FUNCTION IsValidExtension : BOOL
VAR_INPUT
	Extension : I_Extension;
END_VAR

IsValidExtension := Extension <> 0;

END_FUNCTION

(* stored: Version 1.1.0.1, ProductVersion 3.1.4024.12
   POU IsValidExtension: Id {34536ead-6456-0834-1914-3239effc489b}, SpecialFunc None *)
